{attribute 'OPC.UA.DA.JobMethod' := 'JobMethode_HardeningProcess'}
FUNCTION_BLOCK MBS_MR01_AS_HardeningProcess
VAR
	AlwaysTrue : BOOL := TRUE;
	// Used for debugging purposes to display InputArguments of method call
	MethodCall_HardeningProcess : BOOL := FALSE; // used to store InputArg "MethodCall" from Start() method
	ProcessingTime_HardeningProcess : TIME;
	TS_EndschalterEntlastung : BOOL;
	callCounterStart : ULINT; // counts how many times the Start() method has been called
	callCounterCheckState : ULINT; // counts how many times the CheckState() method has been called
	callCounterAbort : ULINT; // counts how many times the Abort() method has been called
	
	// Variables to determine if a job has been started (Start() method has been called) or finished
	jobRunning : BOOL;
	jobFinished : BOOL;

	// State machine variable
	state : UDINT;
	
	//Variablen des FBs
	ResetCall : BOOL;
	MBS_MR01_HardeningProcess : HardeningProcess;
END_VAR
	
VAR_INPUT
	NotAusSignal: BOOL;
	LightSensor_01 : BOOL;
END_VAR

VAR_OUTPUT
	Oven_Ansteuerung : BOOL;
END_VAR

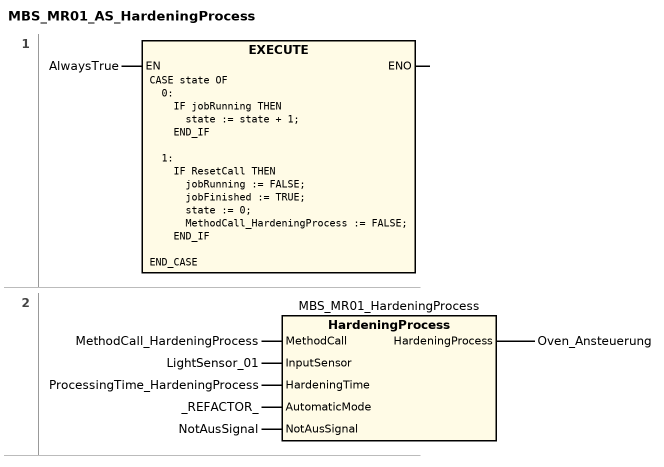
// NETWORK 1
IF AlwaysTrue THEN
    CASE state OF
    	0:
    		IF jobRunning THEN
    			state := state + 1;
    		END_IF
    		
    	1:
    		IF ResetCall THEN
    			jobRunning := FALSE;
    			jobFinished := TRUE;
    			state := 0;
    			MethodCall_HardeningProcess := FALSE;
    		END_IF
    		
    END_CASE
END_IF

// NETWORK 2
MBS_MR01_HardeningProcess(
    MethodCall := MethodCall_HardeningProcess,
    InputSensor := LightSensor_01,
    HardeningTime := ProcessingTime_HardeningProcess,
    AutomaticMode := _REFACTOR_,
    NotAusSignal := NotAusSignal); // HardeningProcess
Oven_Ansteuerung := MBS_MR01_HardeningProcess.HardeningProcess;

{attribute 'TcRpcEnable' := '1'}
METHOD Abort : HRESULT
VAR_INPUT
	hdl : UDINT; // Do not change, used by server.
END_VAR
callCounterAbort := callCounterAbort + 1;
END_METHOD

{attribute 'TcRpcEnable' := '1'}
METHOD CheckState : HRESULT
VAR_INPUT
	hdl : UDINT; // Do not change, used by server.
END_VAR
VAR_OUTPUT
	bBusy : BOOL; // Do not change. Used by server to find out if the job is finished
	
	// List of OutputArguments for OPC UA method, may be customized
	State : BOOL; // Abgeschlossener MethodCall
	MethodCall: BOOL; //Input Recall
END_VAR
callCounterCheckState := callCounterCheckState + 1;
IF NOT jobFinished THEN
	bBusy := TRUE; // job is not finished yet
	CheckState := 0; // no error
ELSE
	bBusy := FALSE; // job is finished
	CheckState := 0; // done, no error occured during execution (OPC UA StatusCode "GOOD")
	jobFinished := FALSE;
	State := ResetCall;
	MethodCall := MethodCall_HardeningProcess;
END_IF
END_METHOD

{attribute 'TcRpcEnable' := '1'}
METHOD Start : HRESULT
VAR_INPUT
	// List of InputArguments for OPC UA method, may be customized
	MethodCall : BOOL; // some description
	ProcessingTime : TIME;
END_VAR
VAR_OUTPUT
	hdl : UDINT; // Do not change, used by server.
END_VAR
callCounterStart := callCounterStart + 1;

MethodCall_HardeningProcess := MethodCall;
ProcessingTime_HardeningProcess := ProcessingTime;

jobRunning := TRUE;
Start := 0; // no error occured, e.g. while parsing the input arguments (0 = OPC UA StatusCode "GOOD")
END_METHOD

END_FUNCTION_BLOCK

(* stored: Version 1.1.0.1, ProductVersion 3.1.4024.15
   POU MBS_MR01_AS_HardeningProcess: Id {0b15150c-e151-4176-8c25-2296b0472d18}, SpecialFunc None
   Method Abort: Id {ab72069d-3514-416d-ad09-b3ef9a8afe82}
   Method CheckState: Id {acc57b30-e5e7-4174-acc1-d8f0d0ddede6}
   Method Start: Id {c968fbcd-5ad0-4e55-ba29-e7a7d198ec23} *)
